// TIA Portal V20 export
// export: Created 2026-09-10T14:33:11.9642249Z, ExportSetting WithDefaults, DisplayName Totally Integrated Automation Portal, DisplayVersion V20, DisplayName TIA Portal Openness, DisplayVersion V20, DisplayName TIA Portal Version Control Interface, DisplayVersion V20, DisplayName STEP 7 Professional, DisplayVersion V20, DisplayName STEP 7 Safety, DisplayVersion V20, DisplayName WinCC Basic/Comfort/Advanced, DisplayVersion V20, DisplayName WinCC Professional, DisplayVersion V20, DisplayName WinCC Unified, DisplayVersion V20
ORGANIZATION_BLOCK "DiagnosticErrorInterrupt"   // OB82, SCL, DiagnosticErrorInterrupt
{ S7_Optimized_Access := 'TRUE' }
VERSION : 0.1
// Called by the CPU when an I/O module reports a diagnostic. Latches Diag_DB.ModuleFault, which FB_ValveLoop turns into HwHealthy[5] and thence HwWord bit 4, driving the existing System_IO_Module_Fault alarm. Deliberately does not decode IO_State - see the body comment.
// stored: IsIECCheckEnabled false, SetENOAutomatically false
   VAR_INPUT
      IO_State : Word;   // IO state of the HW object
      LADDR : HW_ANY;   // Hardware identifier
      Channel : UInt;   // Channel number
      MultiError : Bool;   // =true if more than one error is present
   END_VAR
   VAR_TEMP
      id : UInt;
   END_VAR
BEGIN

   // Called by the CPU when an I/O module raises a diagnostic: its 24 V supply
   // failing, a DQ output short-circuited to L+ or to ground, a parameter error, or
   // a wire break where that is ever enabled. Those diagnostics were switched on
   // across all 36 modules on 2026-09-06 - they ship DISABLED, which is why nothing
   // would have reached this block even if it had existed earlier.
   //
   // WHY THIS BLOCK DOES NOT DECODE #IO_State
   //
   // The same OB fires when a fault APPEARS and again when it GOES AWAY, and
   // #IO_State is what separates the two. Its bit meanings could not be confirmed
   // from any reachable Siemens source, and this block cannot be tested here:
   // PLCSIM does not simulate module-level diagnostics, for the same reason it does
   // not simulate the station events OB86 handles (handoff item 11).
   //
   // Guessing the polarity would risk precisely the failure OB86's own comment
   // warns about - clearing the flag on failure and setting it on recovery, giving
   // a system that reports healthy exactly when it is not. So this block does not
   // guess. ModuleFault LATCHES on any event and clears only via ModuleFaultAck.
   //
   // The worst case is a stale fault sitting after a module has recovered: visible,
   // irritating, and safe. The opposite error is silent. UnexpMove and DirFault
   // already latch for the same reason.
   //
   // Everything is stored RAW and undecoded so the bit meanings can be LEARNED from
   // the real panel rather than guessed now: pull a module and read
   // LastModuleIoState, plug it back in and read it again. Two observations settle
   // what the documentation would not.

   "Diag_DB".ModuleFault := TRUE;

   #id := #LADDR;
   "Diag_DB".LastModuleLaddr := #id;
   "Diag_DB".LastModuleIoState := #IO_State;
   "Diag_DB".LastModuleChannel := #Channel;
   "Diag_DB".LastModuleMultiError := #MultiError;

   // Saturating, not wrapping. An Int rolling past 32767 into negative would read as
   // a different kind of fault to whoever is looking at it, and the exact count that
   // far out says nothing the latched flag has not already said. What the count is
   // genuinely for is spotting a module that is CHATTERING - rising steadily while
   // ModuleFault has never been cleared.
   IF "Diag_DB".ModuleEventCount < 32767 THEN
       "Diag_DB".ModuleEventCount := "Diag_DB".ModuleEventCount + 1;
   END_IF;
END_ORGANIZATION_BLOCK
